Fanuc KAREL source: kt00346.KL

-- PROVISIONAL review KL for V940-1; original PC SHA256 134956b1378f11c4e0fd16f42bd99b1fb16404f11ac31a39e0d510e7a1e2e688
-- Incomplete behavior may be omitted. Consult companion uncertainty JSON. Do not deploy.
PROGRAM KT00346
%NOLOCKGROUP
VAR
  OUT : BOOLEAN
-- UNRESOLVED_DECL H1 type=002017
-- UNRESOLVED_DECL H2 type=002017
BEGIN
  -- V9_ZERO_TABLE_METADATA_HINT layout=0001; no indexed target words; source/name/runtime held
  -- UNRESOLVED_PC offsets 5-19; opcodes 2E,22,9D,33,B4
  -- UNRESOLVED_PC offsets 24-38; opcodes 2E,22,9D,33,B4
  -- UNRESOLVED_PC offsets 43-57; opcodes 2E,22,9D,33,B4
  -- UNRESOLVED_PC offsets 62-76; opcodes 2E,22,9D,33,B4
  -- UNRESOLVED_PC offsets 81-106; opcodes 22,9D,33,B3,22,9D,33,B3,59,23
  -- UNRESOLVED_PC offsets 111-115; opcodes 7F
END KT00346
